TYPE ST_mcAxisStatus :
STRUCT
	bPowerEnabled		:		BOOL; // Power is enabled
	bHomed				:		BOOL; // Homed
	bStandStill			:		BOOL; // Standstill
	bMoving				: 		BOOL; // Moving
	bError				:       BOOL; // Error
END_STRUCT
END_TYPE

(* stored: Version 1.1.0.1, ProductVersion 3.1.4024.6
   DUT ST_mcAxisStatus: Id {52eef8f2-82f7-48c5-a278-bfc275b4b6d4} *)
